# EPICS autosave request: ADApp/Db/simDetector_settings.req
$(P)$(R)GainX
$(P)$(R)GainY
$(P)$(R)GainRed
$(P)$(R)GainGreen
$(P)$(R)GainBlue
$(P)$(R)SimMode
$(P)$(R)PeakStartX
$(P)$(R)PeakStartY
$(P)$(R)PeakNumX
$(P)$(R)PeakNumY
$(P)$(R)PeakStepX
$(P)$(R)PeakStepY
$(P)$(R)PeakWidthX
$(P)$(R)PeakWidthY
$(P)$(R)PeakVariation
$(P)$(R)Noise
files "ADBase_settings.req", P=$(P), R=$(R)
